% RSLogix 500 project P2_DIGITAL FILLING STATION.RSS, saved by version 8.30.00.16 %
PROJECT "PROJECT2"    % processor: Bul.1763 MicroLogix 1100 Series B %

PROGRAM FILES
  LAD 2 "MAIN"  3 rungs
  LAD 3 "IO"  8 rungs
  LAD 4 "CONV CTRL"  9 rungs

DATA FILES
  O0 OUTPUT  4 elements
  I1 INPUT  6 elements
  S2 STATUS  66 elements
  B3 BINARY  5 elements
  T4 TIMER  3 elements
  C5 COUNTER  1 elements
  R6 CONTROL  1 elements
  N7 INTEGER  1 elements
  F8 FLOAT  1 elements

LADDER 2 "MAIN"
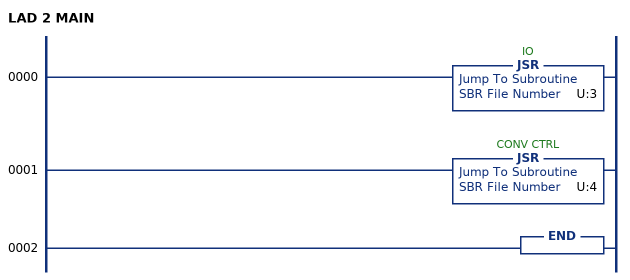
% Rung: 0 %
SOR JSR U:3 EOR
%   U:3  "IO" %
% Rung: 1 %
SOR JSR U:4 EOR
%   U:4  "CONV CTRL" %
% Rung: 2 %
SOR END EOR

LADDER 3 "IO"
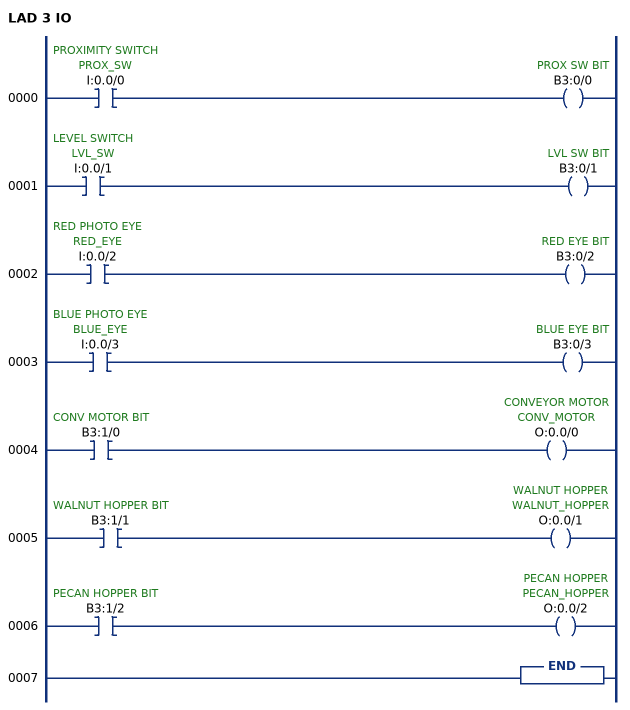
% Rung: 0 %
SOR XIC I:0.0/0 OTE B3:0/0 EOR
%   I:0.0/0  PROX_SW  "PROXIMITY SWITCH" %
%   B3:0/0  "PROX SW BIT" %
% Rung: 1 %
SOR XIC I:0.0/1 OTE B3:0/1 EOR
%   I:0.0/1  LVL_SW  "LEVEL SWITCH" %
%   B3:0/1  "LVL SW BIT" %
% Rung: 2 %
SOR XIC I:0.0/2 OTE B3:0/2 EOR
%   I:0.0/2  RED_EYE  "RED PHOTO EYE" %
%   B3:0/2  "RED EYE BIT" %
% Rung: 3 %
SOR XIC I:0.0/3 OTE B3:0/3 EOR
%   I:0.0/3  BLUE_EYE  "BLUE PHOTO EYE" %
%   B3:0/3  "BLUE EYE BIT" %
% Rung: 4 %
SOR XIC B3:1/0 OTE O:0.0/0 EOR
%   B3:1/0  "CONV MOTOR BIT" %
%   O:0.0/0  CONV_MOTOR  "CONVEYOR MOTOR" %
% Rung: 5 %
SOR XIC B3:1/1 OTE O:0.0/1 EOR
%   B3:1/1  "WALNUT HOPPER BIT" %
%   O:0.0/1  WALNUT_HOPPER  "WALNUT HOPPER" %
% Rung: 6 %
SOR XIC B3:1/2 OTE O:0.0/2 EOR
%   B3:1/2  "PECAN HOPPER BIT" %
%   O:0.0/2  PECAN_HOPPER  "PECAN HOPPER" %
% Rung: 7 %
SOR END EOR

LADDER 4 "CONV CTRL"
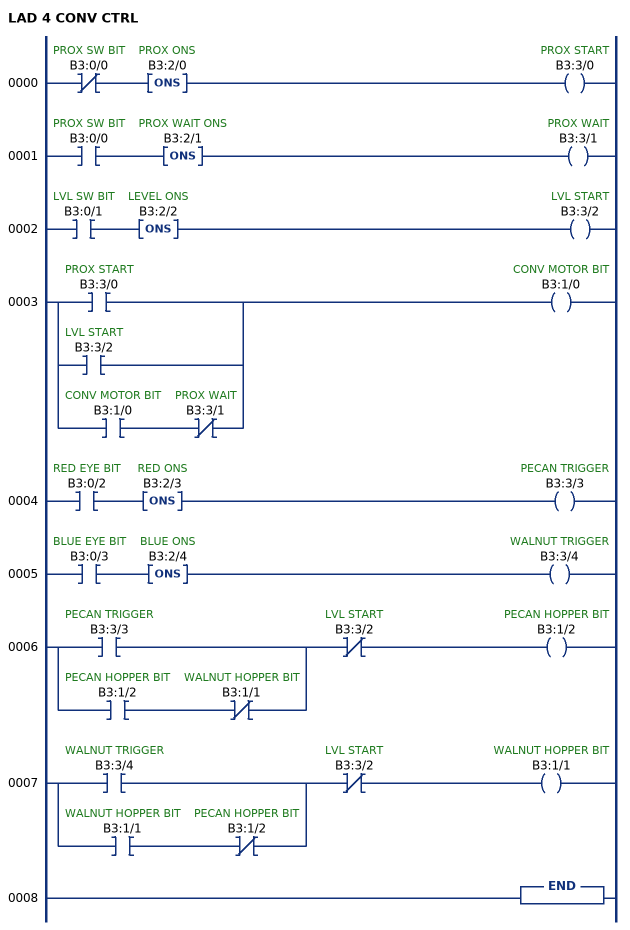
% Rung: 0 %
SOR XIO B3:0/0 ONS B3:2/0 OTE B3:3/0 EOR
%   B3:0/0  "PROX SW BIT" %
%   B3:2/0  "PROX ONS" %
%   B3:3/0  "PROX START" %
% Rung: 1 %
SOR XIC B3:0/0 ONS B3:2/1 OTE B3:3/1 EOR
%   B3:0/0  "PROX SW BIT" %
%   B3:2/1  "PROX WAIT ONS" %
%   B3:3/1  "PROX WAIT" %
% Rung: 2 %
SOR XIC B3:0/1 ONS B3:2/2 OTE B3:3/2 EOR
%   B3:0/1  "LVL SW BIT" %
%   B3:2/2  "LEVEL ONS" %
%   B3:3/2  "LVL START" %
% Rung: 3 %
SOR BST XIC B3:3/0 NXB XIC B3:3/2 NXB XIC B3:1/0 XIO B3:3/1 BND OTE B3:1/0 EOR
%   B3:3/0  "PROX START" %
%   B3:3/2  "LVL START" %
%   B3:1/0  "CONV MOTOR BIT" %
%   B3:3/1  "PROX WAIT" %
% Rung: 4 %
SOR XIC B3:0/2 ONS B3:2/3 OTE B3:3/3 EOR
%   B3:0/2  "RED EYE BIT" %
%   B3:2/3  "RED ONS" %
%   B3:3/3  "PECAN TRIGGER" %
% Rung: 5 %
SOR XIC B3:0/3 ONS B3:2/4 OTE B3:3/4 EOR
%   B3:0/3  "BLUE EYE BIT" %
%   B3:2/4  "BLUE ONS" %
%   B3:3/4  "WALNUT TRIGGER" %
% Rung: 6 %
SOR BST XIC B3:3/3 NXB XIC B3:1/2 XIO B3:1/1 BND XIO B3:3/2 OTE B3:1/2 EOR
%   B3:3/3  "PECAN TRIGGER" %
%   B3:1/2  "PECAN HOPPER BIT" %
%   B3:1/1  "WALNUT HOPPER BIT" %
%   B3:3/2  "LVL START" %
% Rung: 7 %
SOR BST XIC B3:3/4 NXB XIC B3:1/1 XIO B3:1/2 BND XIO B3:3/2 OTE B3:1/1 EOR
%   B3:3/4  "WALNUT TRIGGER" %
%   B3:1/1  "WALNUT HOPPER BIT" %
%   B3:1/2  "PECAN HOPPER BIT" %
%   B3:3/2  "LVL START" %
% Rung: 8 %
SOR END EOR

OTHER DOCUMENTED ADDRESSES
  B3:0  "INPUTS"
  B3:1  "OUTPUTS"
  B3:2  "ONS"
  B3:3  "CONVEYOR"
  T4:0  "PROX DELAY TIMER"
  T4:1  "LVL DELAY TIMER"
  U:2  "IO"
  U:5  "HPR CTRL"

DATA TABLE (non-zero values as saved)
DATA B3
% B3:0 % 0X0000 0X0001 0X0001 0X0000 0X0000
DATA T4
% .PRE .ACC %
% T4:0 % 1 0
